PROGRAM Permissives
VAR
	i : INT := 1;  //for section 1 - 3 
	j : INT := 1; //for charger 1-8
	k : INT := 1; //cap 1- 10
	m : INT := 1; //form cap 1-12
	n : INT := 1; //1-6
	p : INT := 7; //7-12
END_VAR

//Charger summary faults
//Trips_DB.AnySummaryFault = FALSE AND Trips_DB.AnyEstopPressed //add to no fault detected.

//section ready to charge
FOR i := 1 TO 3 BY 1 DO
	IF Trips_DB.NoFaultDetected = TRUE AND //MCP_IO.Charger[1-8].HVisOn AND
		Permissives_DB.AllChargeRelaysClosed = TRUE AND
		LCP.Section[i].Peak.ShortContact1Engaged = FALSE AND
		LCP.Section[i].Peak.ShortContact2Engaged = FALSE AND
		LCP.Section[i].Sust.ShortContact1Engaged = FALSE AND
		LCP.Section[i].Sust.ShortContact2Engaged = FALSE
	THEN
		LCP.Section[i].SystemReadyToCharge := TRUE;	
	ELSE
		LCP.Section[i].SystemReadyToCharge := FALSE;		
	END_IF;
END_FOR;

//Section 4
IF Trips_DB.NoFaultDetected = TRUE AND //MCP_IO.Charger[1-8].HVisOn AND
	Permissives_DB.AllChargeRelaysClosed = TRUE AND
	LCP.Section[4].Form.ShortContact1Engaged = FALSE AND
	LCP.Section[4].Form.ShortContact2Engaged = FALSE AND
	LCP.Section[4].Form.FormTrigShortContactEngaged = FALSE AND
	LCP.Section[4].Form.PreFormTrigShortContactEngaged = FALSE 
	THEN
		LCP.Section[4].SystemReadyToCharge := TRUE;
	ELSE
		LCP.Section[4].SystemReadyToCharge := FALSE;
END_IF;
	
IF LCP.Section[1].SystemReadyToCharge = TRUE AND 
	LCP.Section[2].SystemReadyToCharge = TRUE AND
	LCP.Section[3].SystemReadyToCharge = TRUE AND
	LCP.Section[4].SystemReadyToCharge = TRUE
	THEN
		Permissives_DB.AllSystemsReadytoCharge := TRUE;
		ELSE
			Permissives_DB.AllSystemsReadytoCharge := FALSE;
END_IF


// shorts and unshorts
//Peaking  -- short contacts are NO, so if close is false, it is and unshort is true, then it is not shorted 
FOR i := 1 TO 3 BY 1 DO
	IF LCP.Section[i].Peak.ShortContact1_close = TRUE AND LCP.Section[i].Peak.UnshortContact1_close = FALSE 
		THEN
			LCP.Section[i].Peak.ShortContact1Engaged := TRUE;
		ELSE
			LCP.Section[i].Peak.ShortContact1Engaged := FALSE;
	END_IF;
	
	IF LCP.Section[i].Peak.ShortContact2_close = TRUE AND LCP.Section[i].Peak.UnshortContact2_close = FALSE 
		THEN
			LCP.Section[i].Peak.ShortContact2Engaged := TRUE;
		ELSE
			LCP.Section[i].Peak.ShortContact2Engaged := FALSE;
	END_IF;
	
END_FOR;

//Sustain
FOR i := 1 TO 3 BY 1 DO
	IF LCP.Section[i].Sust.ShortContact1_close = TRUE AND LCP.Section[i].Sust.UnshortContact1_close = FALSE 
		THEN
			LCP.Section[i].Sust.ShortContact1Engaged := TRUE;
		ELSE
			LCP.Section[i].Sust.ShortContact1Engaged := FALSE;
	END_IF;
	
	IF LCP.Section[i].Sust.ShortContact2_close = TRUE AND LCP.Section[i].Sust.UnshortContact2_close = FALSE 
		THEN
			LCP.Section[i].Sust.ShortContact2Engaged := TRUE;
		ELSE
			LCP.Section[i].Sust.ShortContact2Engaged := FALSE;
	END_IF;
	
END_FOR;

//Formation
IF LCP.Section[4].Form.ShortContact1_close = TRUE AND LCP.Section[4].Form.UnshortContact1_close = FALSE
	THEN
		LCP.Section[4].Form.ShortContact1Engaged := TRUE;
	ELSE
		LCP.Section[4].Form.ShortContact1Engaged := FALSE; //might need to clarify on the NC of the short contacts.
END_IF;

IF LCP.Section[4].Form.ShortContact2_close = TRUE AND LCP.Section[4].Form.UnshortContact2_close = FALSE 
	THEN
		LCP.Section[4].Form.ShortContact2Engaged := TRUE;
	ELSE
		LCP.Section[4].Form.ShortContact2Engaged := FALSE; //might need to clarify on the NC of the short contacts.
END_IF;

// form trig short 
IF LCP.Section[4].Form.FormTrigShortContact_close = TRUE AND LCP.Section[4].Form.FormTrigUnShortContact_close = FALSE
	THEN
		LCP.Section[4].Form.FormTrigShortContactEngaged := TRUE;
	ELSE
		LCP.Section[4].Form.FormTrigShortContactEngaged := FALSE;
END_IF
// preform trig short 
IF LCP.Section[4].Form.PreFormTrigShortContact_close = TRUE AND LCP.Section[4].Form.PreFormTrigUnShortContact_close = FALSE
	THEN
		LCP.Section[4].Form.PreFormTrigShortContactEngaged := TRUE;
	ELSE
		LCP.Section[4].Form.PreFormTrigShortContactEngaged := FALSE;
END_IF

//short contacts unknown - This should have never happen
FOR i := 1 TO 3 BY 1 DO
	//Peak
	IF (LCP.Section[i].Peak.ShortContact1_close = TRUE AND LCP.Section[i].Peak.UnShortContact1_close = TRUE) OR 
 		(LCP.Section[i].Peak.ShortContact1_close = FALSE AND LCP.Section[i].Peak.UnShortContact1_close = FALSE)
		THEN
			LCP.Section[i].Peak.ShortContact1unknown := TRUE;
			ELSE
				LCP.Section[i].Peak.ShortContact1unknown := FALSE;
	END_IF;
	
	IF (LCP.Section[i].Peak.ShortContact2_close = TRUE AND LCP.Section[i].Peak.UnShortContact2_close = TRUE) OR 
 		(LCP.Section[i].Peak.ShortContact2_close = FALSE AND LCP.Section[i].Peak.UnShortContact2_close = FALSE)
		THEN
			LCP.Section[i].Peak.ShortContact2unknown := TRUE;
			ELSE
				LCP.Section[i].Peak.ShortContact2unknown := FALSE;
	END_IF;
	//Sust
	IF (LCP.Section[i].Sust.ShortContact1_close = TRUE AND LCP.Section[i].Sust.UnShortContact1_close = TRUE) OR 
 		(LCP.Section[i].Sust.ShortContact1_close = FALSE AND LCP.Section[i].Sust.UnShortContact1_close = FALSE)
		THEN
			LCP.Section[i].Sust.ShortContact1unknown := TRUE;
			ELSE
				LCP.Section[i].Sust.ShortContact1unknown := FALSE;
	END_IF;	
	
	IF (LCP.Section[i].Sust.ShortContact2_close = TRUE AND LCP.Section[i].Sust.UnShortContact2_close = TRUE) OR 
 		(LCP.Section[i].Sust.ShortContact2_close = FALSE AND LCP.Section[i].Sust.UnShortContact2_close = FALSE)
		THEN
			LCP.Section[i].Sust.ShortContact2unknown := TRUE;
			ELSE
				LCP.Section[i].Sust.ShortContact2unknown := FALSE;
	END_IF;	
	
END_FOR;

//Formation
IF (LCP.Section[4].Form.ShortContact1_close = TRUE AND LCP.Section[4].Form.UnShortContact1_close = TRUE) OR 
 	(LCP.Section[4].Form.ShortContact1_close = FALSE AND LCP.Section[4].Form.UnShortContact1_close = FALSE)
	THEN
		LCP.Section[4].Form.ShortContact1unknown := TRUE;
		ELSE
			LCP.Section[4].Form.ShortContact1unknown := FALSE;
END_IF;	
	
IF (LCP.Section[4].Form.ShortContact2_close = TRUE AND LCP.Section[4].Form.UnShortContact2_close = TRUE) OR 
 	(LCP.Section[4].Form.ShortContact2_close = FALSE AND LCP.Section[4].Form.UnShortContact2_close = FALSE)
	THEN
		LCP.Section[4].Form.ShortContact2unknown := TRUE;
		ELSE
			LCP.Section[4].Form.ShortContact2unknown := FALSE;
END_IF;	

IF (LCP.Section[4].Form.FormTrigUnshortContact_close = TRUE AND LCP.Section[4].Form.FormTrigUnshortContact_close = TRUE) OR 
	(LCP.Section[4].Form.FormTrigUnshortContact_close = FALSE AND LCP.Section[4].Form.FormTrigUnshortContact_close = FALSE)
	THEN 
		LCP.Section[4].Form.FormTrigShortContactUnknown := TRUE;
		ELSE
			LCP.Section[4].Form.FormTrigShortContactUnknown := FALSE;
END_IF;

IF (LCP.Section[4].Form.PreFormTrigShortContact_close = TRUE AND LCP.Section[4].Form.PreFormTrigUnShortContact_close = TRUE) OR
	(LCP.Section[4].Form.PreFormTrigShortContact_close = FALSE AND LCP.Section[4].Form.PreFormTrigUnShortContact_close = FALSE)
	THEN
		LCP.Section[4].Form.PreFormTrigShortContactUnknown := TRUE;
		ELSE
			LCP.Section[4].Form.PreFormTrigShortContactUnknown := FALSE;
END_IF;
	
// any short contact in unknown state?
IF LCP.Section[1].Peak.ShortContact1unknown = FALSE AND 
	LCP.Section[1].Peak.ShortContact2unknown = FALSE AND
	LCP.Section[2].Peak.ShortContact1unknown = FALSE AND
	LCP.Section[2].Peak.ShortContact2unknown = FALSE AND
	LCP.Section[3].Peak.ShortContact1unknown = FALSE AND
	LCP.Section[3].Peak.ShortContact2unknown = FALSE AND
	LCP.Section[1].Sust.ShortContact1unknown = FALSE AND
	LCP.Section[1].Sust.ShortContact2unknown = FALSE AND
	LCP.Section[2].Sust.ShortContact1unknown = FALSE AND 
	LCP.Section[2].Sust.ShortContact2unknown = FALSE AND
	LCP.Section[3].Sust.ShortContact1unknown = FALSE AND 
	LCP.Section[3].Sust.ShortContact2unknown = FALSE AND
	LCP.Section[4].Form.ShortContact1unknown = FALSE AND
	LCP.Section[4].Form.ShortContact2unknown = FALSE AND 
	LCP.Section[4].Form.FormTrigShortContactUnknown = FALSE AND //
	LCP.Section[4].Form.PreFormTrigShortContactUnknown = FALSE //
	THEN
		Permissives_DB.NoShortingUnknowns := TRUE;
	ELSE
		Permissives_DB.NoShortingUnknowns := FALSE;
END_IF;


//any short contact engaged

IF LCP.Section[1].Peak.ShortContact1Engaged = TRUE AND 
	LCP.Section[1].Peak.ShortContact2Engaged = TRUE AND
	LCP.Section[2].Peak.ShortContact1Engaged = TRUE AND
	LCP.Section[2].Peak.ShortContact2Engaged = TRUE AND
	LCP.Section[3].Peak.ShortContact1Engaged = TRUE AND
	LCP.Section[3].Peak.ShortContact2Engaged = TRUE AND
	LCP.Section[1].Sust.ShortContact1Engaged = TRUE AND
	LCP.Section[1].Sust.ShortContact2Engaged = TRUE AND
	LCP.Section[2].Sust.ShortContact1Engaged = TRUE AND 
	LCP.Section[2].Sust.ShortContact2Engaged = TRUE AND
	LCP.Section[3].Sust.ShortContact1Engaged = TRUE AND 
	LCP.Section[3].Sust.ShortContact2Engaged = TRUE AND
	LCP.Section[4].Form.ShortContact1Engaged = TRUE AND
	LCP.Section[4].Form.ShortContact2Engaged = TRUE AND 
	LCP.Section[4].Form.FormTrigShortContactEngaged = TRUE AND //
	LCP.Section[4].Form.PreFormTrigShortContactEngaged = TRUE //
	THEN
		Permissives_DB.AllShortContactEngaged := TRUE;
	ELSE 
		Permissives_DB.AllShortContactEngaged := FALSE;	
END_IF;

//All charger inhibited
IF (MCP_IO.Charger[1].inhibited = TRUE OR Recipe.PeakSupplyEN = FALSE) AND
	(MCP_IO.Charger[2].inhibited = TRUE OR Recipe.PeakSupplyEN = FALSE) AND
	(MCP_IO.Charger[3].inhibited = TRUE OR Recipe.PeakSupplyEN = FALSE) //AND
	//(MCP_IO.Charger[4].inhibited = TRUE OR Recipe.SustSupplyEN = FALSE) AND
	//(MCP_IO.Charger[5].inhibited = TRUE OR Recipe.SustSupplyEN = FALSE) AND
	//(MCP_IO.Charger[6].inhibited = TRUE OR Recipe.SustSupplyEN = FALSE) AND
	//(MCP_IO.Charger[7].inhibited = TRUE OR Recipe.FormSupplyEN = FALSE) AND
	//(MCP_IO.Charger[8].inhibited = TRUE OR Recipe.FormSupplyEN = FALSE) 
	THEN
		Permissives_DB.AllChargerInhibited := TRUE;
		ELSE
			Permissives_DB.AllChargerInhibited := FALSE;
END_IF;

//All charger HV ON
IF (MCP_IO.Charger[1].HV_isON = TRUE OR Recipe.PeakSupplyEN = FALSE) AND
	(MCP_IO.Charger[2].HV_isON = TRUE OR Recipe.PeakSupplyEN = FALSE) AND
	(MCP_IO.Charger[3].HV_isON = TRUE OR Recipe.PeakSupplyEN = FALSE) (*AND
	(MCP_IO.Charger[4].HV_isON = TRUE OR Recipe.SustSupplyEN = FALSE) AND
	(MCP_IO.Charger[5].HV_isON = TRUE OR Recipe.SustSupplyEN = FALSE) AND
	(MCP_IO.Charger[6].HV_isON = TRUE OR Recipe.SustSupplyEN = FALSE) AND
	(MCP_IO.Charger[7].HV_isON = TRUE OR Recipe.FormSupplyEN = FALSE) AND
	(MCP_IO.Charger[8].HV_isON = TRUE OR Recipe.FormSupplyEN = FALSE) AND
	(MCP_IO.GLS3_hvON = TRUE OR Recipe.PFormSupplyEN = FALSE)*)
	THEN
		Permissives_DB.AllChargerHVisON := TRUE;
		ELSE
			Permissives_DB.AllChargerHVisON := FALSE;
END_IF;

//peaking ch hv on
IF MCP_IO.Charger[1].HV_isON = TRUE AND 
	MCP_IO.Charger[2].HV_isON = TRUE AND 
	MCP_IO.Charger[3].HV_isON = TRUE 
	THEN
		Permissives_DB.AllPeakChargerHVisON := TRUE;
		ELSE
			Permissives_DB.AllPeakChargerHVisON := FALSE;
END_IF
//sustain ch hv on
(*IF MCP_IO.Charger[4].HV_isON = TRUE AND 
	MCP_IO.Charger[5].HV_isON = TRUE AND 
	MCP_IO.Charger[6].HV_isON = TRUE 
	THEN
		Permissives_DB.AllSustChargerHVisON := TRUE;
		ELSE
			Permissives_DB.AllSustChargerHVisON := FALSE;
END_IF
//Form ch hv on
IF MCP_IO.Charger[7].HV_isON = TRUE AND 
	MCP_IO.Charger[8].HV_isON = TRUE  
	THEN
		Permissives_DB.AllFormChargerHVisON := TRUE;
		ELSE
			Permissives_DB.AllFormChargerHVisON := FALSE;
END_IF*)
//peaking ch inhibit
IF MCP_IO.Charger[1].inhibited = TRUE AND 
	MCP_IO.Charger[2].inhibited = TRUE AND 
	MCP_IO.Charger[3].inhibited = TRUE 
	THEN
		Permissives_DB.AllPeakChargerInhibited := TRUE;
		ELSE
			Permissives_DB.AllPeakChargerInhibited := FALSE;
END_IF
//sust ch inhibit
(*IF MCP_IO.Charger[4].inhibited = TRUE AND 
	MCP_IO.Charger[5].inhibited = TRUE AND 
	MCP_IO.Charger[6].inhibited = TRUE 
	THEN
		Permissives_DB.AllSustChargerInhibited := TRUE;
		ELSE
			Permissives_DB.AllSustChargerInhibited := FALSE;
END_IF
//form ch inhibit
IF MCP_IO.Charger[7].inhibited = TRUE AND 
	MCP_IO.Charger[8].inhibited = TRUE
	THEN
		Permissives_DB.AllFormChargerInhibited := TRUE;
		ELSE
			Permissives_DB.AllFormChargerInhibited := FALSE;
END_IF*)

IF (MCP_IO.Charger[1].EndOfCharge = TRUE OR Recipe.PeakSupplyEN = FALSE) AND
	(MCP_IO.Charger[2].EndOfCharge = TRUE OR Recipe.PeakSupplyEN = FALSE) AND
	(MCP_IO.Charger[3].EndOfCharge = TRUE OR Recipe.PeakSupplyEN = FALSE) (*AND
	(MCP_IO.Charger[4].EndOfCharge = TRUE OR Recipe.SustsupplyEN = FALSE) AND
	(MCP_IO.Charger[5].EndOfCharge = TRUE OR Recipe.SustsupplyEN = FALSE) AND
	(MCP_IO.Charger[6].EndOfCharge = TRUE OR Recipe.SustsupplyEN = FALSE) AND
	(MCP_IO.Charger[7].EndOfCharge = TRUE OR Recipe.FormSupplyEN = FALSE) AND
	(MCP_IO.Charger[8].EndOfCharge = TRUE OR Recipe.FormSupplyEN = FALSE) *)
	THEN 
		Permissives_DB.AllChargerEOC := TRUE;
		ELSE
			Permissives_DB.AllChargerEOC := FALSE;
END_IF

//all peaking charg
IF LCP.Section[1].Peak.ChargeRelay1_close = TRUE AND
	LCP.Section[1].Peak.ChargeRelay2_close = TRUE AND
	LCP.Section[2].Peak.ChargeRelay1_close = TRUE AND
	LCP.Section[2].Peak.ChargeRelay2_close = TRUE AND
	LCP.Section[3].Peak.ChargeRelay1_close = TRUE AND
	LCP.Section[3].Peak.ChargeRelay2_close = TRUE 
	THEN
		Permissives_DB.AllPeakChargeRlyClose := TRUE;
		ELSE
			Permissives_DB.AllPeakChargeRlyClose := FALSE;
END_IF

//all sust charge
IF LCP.Section[1].Sust.ChargeRelay1_close = TRUE AND
	LCP.Section[1].Sust.ChargeRelay2_close = TRUE AND
	LCP.Section[2].Sust.ChargeRelay1_close = TRUE AND
	LCP.Section[2].Sust.ChargeRelay2_close = TRUE AND
	LCP.Section[3].Sust.ChargeRelay1_close = TRUE AND
	LCP.Section[3].Sust.ChargeRelay2_close = TRUE 
	THEN
		Permissives_DB.AllSustChargeRlyClose := TRUE;
		ELSE
			Permissives_DB.AllSustChargeRlyClose := FALSE;
END_IF
//all form charge
IF	LCP.Section[4].Form.ChargeRelay1_close = TRUE AND
	LCP.Section[4].Form.ChargeRelay2_close = TRUE 
	THEN
		Permissives_DB.AllFormChargeRlyClose := TRUE;
		ELSE
			Permissives_DB.AllFormChargeRlyClose := FALSE;
END_IF

//all peak dump
IF LCP.Section[1].Peak.DumpRelay1_close = TRUE AND
	LCP.Section[1].Peak.DumpRelay2_close = TRUE AND
	LCP.Section[2].Peak.DumpRelay1_close = TRUE AND
	LCP.Section[2].Peak.DumpRelay2_close = TRUE AND
	LCP.Section[3].Peak.DumpRelay1_close = TRUE AND
	LCP.Section[3].Peak.DumpRelay2_close = TRUE 
	THEN
		Permissives_DB.AllPeakDumpRlyOpen := FALSE;
		ELSE
			Permissives_DB.AllPeakDumpRlyOpen := TRUE;
END_IF
//all sust dump
IF LCP.Section[1].Sust.DumpRelay1_close = TRUE AND
	LCP.Section[1].Sust.DumpRelay2_close = TRUE AND
	LCP.Section[2].Sust.DumpRelay1_close = TRUE AND
	LCP.Section[2].Sust.DumpRelay2_close = TRUE AND
	LCP.Section[3].Sust.DumpRelay1_close = TRUE AND
	LCP.Section[3].Sust.DumpRelay2_close = TRUE 
	THEN
		Permissives_DB.AllSustDumpRlyOpen := FALSE;
		ELSE
			Permissives_DB.AllSustDumpRlyOpen := TRUE;
END_IF
//all form dump
IF LCP.Section[4].Form.DumpRelay1_close = TRUE AND
	LCP.Section[4].Form.DumpRelay2_close = TRUE 
	THEN
		Permissives_DB.AllFormDumpRlyOpen := FALSE;
		ELSE
			Permissives_DB.AllFormDumpRlyOpen := TRUE;
END_IF
// GLS 1 & 2 can use raw input bit.

//section 1 charge
IF LCP.Section[1].Peak.ChargeRelay1_close = TRUE AND
	LCP.Section[1].Peak.ChargeRelay2_close = TRUE AND
	LCP.Section[1].Sust.ChargeRelay1_close = TRUE AND
	LCP.Section[1].Sust.ChargeRelay2_close = TRUE 
	THEN
		Permissives_DB.AllSection1ChargeRlyClose := TRUE;
		ELSE
			Permissives_DB.AllSection1ChargeRlyClose := FALSE;
END_IF;
//section 2 charge
IF LCP.Section[2].Peak.ChargeRelay1_close = TRUE AND
	LCP.Section[2].Peak.ChargeRelay2_close = TRUE AND
	LCP.Section[2].Sust.ChargeRelay1_close = TRUE AND
	LCP.Section[2].Sust.ChargeRelay2_close = TRUE 
	THEN
		Permissives_DB.AllSection2ChargeRlyClose := TRUE;
		ELSE
			Permissives_DB.AllSection2ChargeRlyClose := FALSE;
END_IF;
//section 3 charge
IF LCP.Section[3].Peak.ChargeRelay1_close = TRUE AND
	LCP.Section[3].Peak.ChargeRelay2_close = TRUE AND
	LCP.Section[3].Sust.ChargeRelay1_close = TRUE AND
	LCP.Section[3].Sust.ChargeRelay2_close = TRUE 
	THEN
		Permissives_DB.AllSection3ChargeRlyClose := TRUE;
		ELSE
			Permissives_DB.AllSection3ChargeRlyClose := FALSE;
END_IF;
//section 4 charge
IF	LCP.Section[4].Form.ChargeRelay1_close = TRUE AND
	LCP.Section[4].Form.ChargeRelay2_close = TRUE AND						
	LCP.Section[4].Form.PreFormChargeRly_close = TRUE AND
	LCP.Section[4].Form.FormTrigChargeRly_close = TRUE AND
	LCP.Section[4].Form.PreFormTrigChargeRly_close = TRUE
	THEN
		Permissives_DB.AllSection4ChargeRlyClose := TRUE;
		ELSE
			Permissives_DB.AllSection4ChargeRlyClose := FALSE;
END_IF
	
//All charge relay close
IF ((LCP.Section[1].Peak.ChargeRelay1_close = TRUE OR Recipe.PeakSupplyEN = FALSE)AND
	(LCP.Section[1].Peak.ChargeRelay2_close = TRUE OR Recipe.PeakSupplyEN = FALSE)AND
	(LCP.Section[1].Sust.ChargeRelay1_close = TRUE OR Recipe.SustSupplyEN = FALSE)AND
	(LCP.Section[1].Sust.ChargeRelay2_close = TRUE OR Recipe.SustSupplyEN = FALSE)AND
	(LCP.Section[2].Peak.ChargeRelay1_close = TRUE OR Recipe.PeakSupplyEN = FALSE)AND
	(LCP.Section[2].Peak.ChargeRelay2_close = TRUE OR Recipe.PeakSupplyEN = FALSE)AND
	(LCP.Section[2].Sust.ChargeRelay1_close = TRUE OR Recipe.SustSupplyEN = FALSE)AND
	(LCP.Section[2].Sust.ChargeRelay2_close = TRUE OR Recipe.SustSupplyEN = FALSE)AND
	(LCP.Section[3].Peak.ChargeRelay1_close = TRUE OR Recipe.PeakSupplyEN = FALSE)AND
	(LCP.Section[3].Peak.ChargeRelay2_close = TRUE OR Recipe.PeakSupplyEN = FALSE)AND
	(LCP.Section[3].Sust.ChargeRelay1_close = TRUE OR Recipe.SustSupplyEN = FALSE)AND
	(LCP.Section[3].Sust.ChargeRelay2_close = TRUE OR Recipe.SustSupplyEN = FALSE)AND
	
	(LCP.Section[4].Form.ChargeRelay1_close = TRUE OR Recipe.FormSupplyEN = FALSE)AND
	(LCP.Section[4].Form.ChargeRelay2_close = TRUE OR Recipe.FormSupplyEN = FALSE)AND						
	(LCP.Section[4].Form.PreFormChargeRly_close = TRUE OR Recipe.PFormSupplyEN = FALSE)AND
	(LCP.Section[4].Form.FormTrigChargeRly_close = TRUE  OR Recipe.FormSupplyEN = FALSE)AND
	(LCP.Section[4].Form.PreFormTrigChargeRly_close = TRUE OR Recipe.PFormSupplyEN = FALSE)) OR HMI_DB.AllChargeRelayCloseBP = TRUE //admin bypass 
	THEN
		Permissives_DB.AllChargeRelaysClosed := TRUE;
	ELSE
		Permissives_DB.AllChargeRelaysClosed := FALSE;
END_IF;

//section 1 dump
IF LCP.Section[1].Peak.DumpRelay1_close = FALSE AND
	LCP.Section[1].Peak.DumpRelay2_close = FALSE AND
	LCP.Section[1].Sust.DumpRelay1_close = FALSE AND
	LCP.Section[1].Sust.DumpRelay2_close = FALSE
	THEN
		Permissives_DB.AllSection1DumpRlyOpen := TRUE;
		ELSE
			Permissives_DB.AllSection1DumpRlyOpen := FALSE;
END_IF
//section 2 dump
IF LCP.Section[2].Peak.DumpRelay1_close = FALSE AND
	LCP.Section[2].Peak.DumpRelay2_close = FALSE AND
	LCP.Section[2].Sust.DumpRelay1_close = FALSE AND
	LCP.Section[2].Sust.DumpRelay2_close = FALSE
	THEN
		Permissives_DB.AllSection2DumpRlyOpen := TRUE;
		ELSE
			Permissives_DB.AllSection2DumpRlyOpen := FALSE;
END_IF
//section 3 dump
IF LCP.Section[3].Peak.DumpRelay1_close = FALSE AND
	LCP.Section[3].Peak.DumpRelay2_close = FALSE AND
	LCP.Section[3].Sust.DumpRelay1_close = FALSE AND
	LCP.Section[3].Sust.DumpRelay2_close = FALSE
	THEN
		Permissives_DB.AllSection3DumpRlyOpen := TRUE;
		ELSE
			Permissives_DB.AllSection3DumpRlyOpen := FALSE;
END_IF
//section 4 dump
IF 	LCP.Section[4].Form.DumpRelay1_close = FALSE AND
	LCP.Section[4].Form.DumpRelay2_close = FALSE AND						
	LCP.Section[4].Form.PreFormDumpRly_close = FALSE AND
	LCP.Section[4].Form.FormTrigDumpRly1_close = FALSE AND
	LCP.Section[4].Form.PreFormTrigDumpRly1_close = FALSE
	THEN
		Permissives_DB.AllSection4DumpRlyOpen := TRUE;
		ELSE
			Permissives_DB.AllSection4DumpRlyOpen := FALSE;
END_IF

//All Dump relays open  ******
IF (LCP.Section[1].Peak.DumpRelay1_close = FALSE AND
	LCP.Section[1].Peak.DumpRelay2_close = FALSE AND
	LCP.Section[1].Sust.DumpRelay1_close = FALSE AND
	LCP.Section[1].Sust.DumpRelay2_close = FALSE AND
	LCP.Section[2].Peak.DumpRelay1_close = FALSE AND
	LCP.Section[2].Peak.DumpRelay2_close = FALSE AND
	LCP.Section[2].Sust.DumpRelay1_close = FALSE AND
	LCP.Section[2].Sust.DumpRelay2_close = FALSE AND
	LCP.Section[3].Peak.DumpRelay1_close = FALSE AND
	LCP.Section[3].Peak.DumpRelay2_close = FALSE AND
	LCP.Section[3].Sust.DumpRelay1_close = FALSE AND
	LCP.Section[3].Sust.DumpRelay2_close = FALSE AND
	
	LCP.Section[4].Form.DumpRelay1_close = FALSE AND
	LCP.Section[4].Form.DumpRelay2_close = FALSE AND						
	LCP.Section[4].Form.PreFormDumpRly_close = FALSE AND
	LCP.Section[4].Form.FormTrigDumpRly1_close = FALSE AND
	LCP.Section[4].Form.PreFormTrigDumpRly1_close = FALSE) OR HMI_DB.AllDumpRelaysOpenBP = TRUE //admin bypass 
	THEN
		Permissives_DB.AllDumpRelaysOpen := TRUE;
	ELSE
		Permissives_DB.AllDumpRelaysOpen := FALSE;
END_IF;
//check for cap voltage for fully discharged
FOR i := 1 TO 3 BY 1 DO
	//peak
	FOR k := 1 TO 10 BY 1 DO
		IF LCP.Section[i].Peak.Cap[k].voltageFeedback <= 10 THEN 
			LCP.Section[i].Peak.Cap[k].CapDischaged := TRUE;
			ELSE
				LCP.Section[i].Peak.Cap[k].CapDischaged := FALSE;
		END_IF;
		//check for cap fully charged*************************
		IF LCP.Section[i].Peak.Cap[k].voltageFeedback >= Setpoints.TDKLoad[i].RequiredChargedV THEN 
			LCP.Section[i].Peak.Cap[k].CapfullyCharged := TRUE;
			ELSE
				LCP.Section[i].Peak.Cap[k].CapfullyCharged := FALSE;
		END_IF;
	END_FOR;
	//sus
	IF LCP.Section[i].Sust.Cap[1].voltageFeedback <= 10 THEN
		LCP.Section[i].Sust.Cap[1].CapDischaged := TRUE;
		ELSE
			LCP.Section[i].Sust.Cap[1].CapDischaged := FALSE;
	END_IF;
	//check fo cap fully charged
	IF LCP.Section[i].Sust.Cap[1].voltageFeedback >= Setpoints.TDKLoad[i+3].RequiredChargedV THEN
		LCP.Section[i].Sust.Cap[1].CapfullyCharged := TRUE;
		ELSE
			LCP.Section[i].Sust.Cap[1].CapfullyCharged := FALSE;
	END_IF;
	
	IF LCP.Section[i].Sust.Cap[2].voltageFeedback <= 10 THEN
		LCP.Section[i].Sust.Cap[2].CapDischaged := TRUE;
		ELSE
			LCP.Section[i].Sust.Cap[2].CapDischaged := FALSE;
	END_IF;
	//check for cap fully charged
	IF LCP.Section[i].Sust.Cap[2].voltageFeedback >= Setpoints.TDKLoad[i+3].RequiredChargedV THEN
		LCP.Section[i].Sust.Cap[2].CapfullyCharged := TRUE;
		ELSE
			LCP.Section[i].Sust.Cap[2].CapfullyCharged := FALSE;
	END_IF;
END_FOR;
// form
FOR m := 1 TO 12 BY 1 DO
	IF LCP.Section[4].Form.Cap[m].voltageFeedback <= 10 THEN
		LCP.Section[4].Form.Cap[m].CapDischaged := TRUE;
		ELSE
			LCP.Section[4].Form.Cap[m].CapDischaged := FALSE;
	END_IF;
END_FOR;

//check for cap fully charged
FOR n := 1 TO 6 BY 1 DO 
	IF LCP.Section[4].Form.Cap[n].voltageFeedback >= Setpoints.TDKLoad[7].RequiredChargedV THEN
		LCP.Section[4].Form.Cap[n].CapfullyCharged := TRUE;
		ELSE
			LCP.Section[4].Form.Cap[n].CapfullyCharged := FALSE;
	END_IF;		
END_FOR

FOR p := 7 TO 12 BY 1 DO 
	IF LCP.Section[4].Form.Cap[p].voltageFeedback >= Setpoints.TDKLoad[8].RequiredChargedV THEN
		LCP.Section[4].Form.Cap[p].CapfullyCharged := TRUE;
		ELSE
			LCP.Section[4].Form.Cap[p].CapfullyCharged := FALSE;
	END_IF;		
END_FOR

//preform
IF LCP.Section[4].PreFormCapVoltageFeedback <= 10 THEN
	LCP.Section[4].PreFormCapDischarged := TRUE;
	ELSE
		LCP.Section[4].PreFormCapDischarged := FALSE;
END_IF

//preform
IF LCP.Section[4].PreFormCapVoltageFeedback >= Setpoints.GLSLoad.RequiredChargedV THEN
	LCP.Section[4].PreFormCapFullyChaged := TRUE;
	ELSE
		LCP.Section[4].PreFormCapFullyChaged := FALSE;
END_IF


//all caps discharge condition
FOR i := 1 TO 3 BY 1 DO
	IF LCP.Section[i].Peak.Cap[1].CapDischaged = TRUE AND
		LCP.Section[i].Peak.Cap[2].CapDischaged = TRUE AND
		LCP.Section[i].Peak.Cap[3].CapDischaged = TRUE AND
		LCP.Section[i].Peak.Cap[4].CapDischaged = TRUE AND
		LCP.Section[i].Peak.Cap[5].CapDischaged = TRUE AND
		LCP.Section[i].Peak.Cap[6].CapDischaged = TRUE AND
		LCP.Section[i].Peak.Cap[7].CapDischaged = TRUE AND
		LCP.Section[i].Peak.Cap[8].CapDischaged = TRUE AND
		LCP.Section[i].Peak.Cap[9].CapDischaged = TRUE AND
		LCP.Section[i].Peak.Cap[10].CapDischaged = TRUE AND
		LCP.Section[i].Sust.Cap[1].CapDischaged = TRUE AND
		LCP.Section[i].Sust.Cap[2].CapDischaged = TRUE
		THEN
			LCP.Section[i].AllCapsDischarged := TRUE; 
		ELSE
			LCP.Section[i].AllCapsDischarged := FALSE; 
	END_IF;
	
	//all caps fully charged 
	IF LCP.Section[i].Peak.Cap[1].CapFullyCharged = TRUE AND
		LCP.Section[i].Peak.Cap[2].CapFullyCharged = TRUE AND
		LCP.Section[i].Peak.Cap[3].CapFullyCharged = TRUE AND
		LCP.Section[i].Peak.Cap[4].CapFullyCharged = TRUE AND
		LCP.Section[i].Peak.Cap[5].CapFullyCharged = TRUE AND
		LCP.Section[i].Peak.Cap[6].CapFullyCharged = TRUE AND
		LCP.Section[i].Peak.Cap[7].CapFullyCharged = TRUE AND
		LCP.Section[i].Peak.Cap[8].CapFullyCharged = TRUE AND
		LCP.Section[i].Peak.Cap[9].CapFullyCharged = TRUE AND
		LCP.Section[i].Peak.Cap[10].CapFullyCharged = TRUE AND
		LCP.Section[i].Sust.Cap[1].CapFullyCharged = TRUE AND
		LCP.Section[i].Sust.Cap[2].CapFullyCharged = TRUE
		THEN
			LCP.Section[i].AllCapsFullyCharged := TRUE;
		ELSE
			LCP.Section[i].AllCapsFullyCharged := FALSE;
	END_IF
END_FOR
//form caps 
IF LCP.Section[4].Form.Cap[1].CapDischaged = TRUE AND
	LCP.Section[4].Form.Cap[2].CapDischaged = TRUE AND
	LCP.Section[4].Form.Cap[3].CapDischaged = TRUE AND
	LCP.Section[4].Form.Cap[4].CapDischaged = TRUE AND
	LCP.Section[4].Form.Cap[5].CapDischaged = TRUE AND
	LCP.Section[4].Form.Cap[6].CapDischaged = TRUE AND
	LCP.Section[4].Form.Cap[7].CapDischaged = TRUE AND
	LCP.Section[4].Form.Cap[8].CapDischaged = TRUE AND
	LCP.Section[4].Form.Cap[9].CapDischaged = TRUE AND
	LCP.Section[4].Form.Cap[10].CapDischaged = TRUE AND
	LCP.Section[4].Form.Cap[11].CapDischaged = TRUE AND
	LCP.Section[4].Form.Cap[12].CapDischaged = TRUE AND 
	LCP.Section[4].PreFormCapDischarged = TRUE
	THEN 
		LCP.Section[4].AllCapsDischarged := TRUE;
	ELSE
		LCP.Section[4].AllCapsDischarged := FALSE;	
END_IF
//checking for caps fully charged
IF LCP.Section[4].Form.Cap[1].CapFullyCharged = TRUE AND
	LCP.Section[4].Form.Cap[2].CapFullyCharged = TRUE AND
	LCP.Section[4].Form.Cap[3].CapFullyCharged = TRUE AND
	LCP.Section[4].Form.Cap[4].CapFullyCharged = TRUE AND
	LCP.Section[4].Form.Cap[5].CapFullyCharged = TRUE AND
	LCP.Section[4].Form.Cap[6].CapFullyCharged = TRUE AND
	LCP.Section[4].Form.Cap[7].CapFullyCharged = TRUE AND
	LCP.Section[4].Form.Cap[8].CapFullyCharged = TRUE AND
	LCP.Section[4].Form.Cap[9].CapFullyCharged = TRUE AND
	LCP.Section[4].Form.Cap[10].CapFullyCharged = TRUE AND
	LCP.Section[4].Form.Cap[11].CapFullyCharged = TRUE AND
	LCP.Section[4].Form.Cap[12].CapFullyCharged = TRUE AND
	LCP.Section[4].PreFormCapFullyChaged = TRUE
	THEN
		LCP.Section[4].AllCapsFullyCharged := TRUE;
	ELSE
		LCP.Section[4].AllCapsFullyCharged := FALSE;
END_IF

//all capps fully charged
IF LCP.Section[1].AllCapsFullyCharged = TRUE AND
	LCP.Section[2].AllCapsFullyCharged = TRUE AND
	LCP.Section[3].AllCapsFullyCharged = TRUE AND
	LCP.Section[4].AllCapsFullyCharged = TRUE 
	THEN
		Permissives_DB.AllSectCapsFullyCharged := TRUE;
	ELSE
		Permissives_DB.AllSectCapsFullyCharged := FALSE;
END_IF

IF LCP.Section[1].AllCapsDischarged = TRUE AND
	LCP.Section[2].AllCapsDischarged = TRUE AND
	LCP.Section[3].AllCapsDischarged = TRUE AND
	LCP.Section[4].AllCapsDischarged = TRUE 
	THEN 
		Permissives_DB.AllSectCapsDischarged := TRUE;
	ELSE
		Permissives_DB.AllSectCapsDischarged := FALSE;
END_IF


//no loss in interlock pneumatic pressure

IF (LCP.Section[1].LossPneumaticPressure = FALSE AND
	LCP.Section[2].LossPneumaticPressure = FALSE AND
	LCP.Section[3].LossPneumaticPressure = FALSE AND
	LCP.Section[4].LossPneumaticPressure = FALSE) OR HMI_DB.InterlockPressureLossBP = TRUE 
	THEN
		Permissives_DB.NoInterlockPressureLoss := TRUE;
		ELSE
			Permissives_DB.NoInterlockPressureLoss := FALSE;
END_IF;
	
IF (Permissives_DB.NoShortingUnknowns = TRUE AND
	Trips_DB.AllDCpsuOK = TRUE AND
	Trips_DB.CageEStopCircuitBroken = FALSE AND
	Trips_DB.AnyChargerOverTemp = FALSE AND
	Trips_DB.AnyEstopPressed = FALSE AND
	Trips_DB.AnyChargerInterlockOpen = FALSE AND
	Permissives_DB.NoInterlockPressureLoss = TRUE) OR HMI_DB.SafetyOKBP = TRUE // admin bypass 
	THEN
		Permissives_DB.SafetyOK := TRUE;
		ELSE
			Permissives_DB.SafetyOK := FALSE;
END_IF;

IF i > 3 THEN
	i := 1;
END_IF;

IF j > 8 THEN
	j := 1;
END_IF;

IF k > 10 THEN
	k := 1;
END_IF;

IF m > 12 THEN
	m := 1;
END_IF;

IF n > 6 THEN
	n := 1;
END_IF;

IF p > 12 THEN
	p := 7;
END_IF;

END_PROGRAM

(* stored: Version 1.1.0.1, ProductVersion 3.1.4024.11
   POU Permissives: Id {a037c57d-7935-4b17-bb0a-42e72a6c09c9}, SpecialFunc None *)
